// TIA Portal V18 export
// export: Created 2026-06-12T02:00:00Z, ExportSetting WithDefaults, DisplayName Totally Integrated Automation Portal, DisplayVersion V18, DisplayName TIA Portal Openness, DisplayVersion V18
TagTable "AI_B4_Tags"
  AI_B4_Daq_C : Real  (PLC tag AI_B4_Daq_C, HMI_Connection_1, 1 s)   // COUNT 0-100
  AI_B4_TPH_Total : Real  (PLC tag AI_B4_TPH_Total, HMI_Connection_1, 1 s)   // FLOW 100-200 T/h
  AI_B4_KG_CM_Main : Real  (PLC tag AI_B4_KG_CM_Main, HMI_Connection_1, 1 s)   // PRESSURE 7-8 kg/cm2
  AI_B4_DRM_LVL1 : Real  (PLC tag AI_B4_DRM_LVL1, HMI_Connection_1, 1 s)   // LEVEL 30-80 %
  AI_B4_DRM_LVL2 : Real  (PLC tag AI_B4_DRM_LVL2, HMI_Connection_1, 1 s)   // LEVEL 30-80 %
  AI_B4_MW_Output : Real  (PLC tag AI_B4_MW_Output, HMI_Connection_1, 1 s)   // COUNT 0-50 MW
  AI_B4_KG_CM_2 : Real  (PLC tag AI_B4_KG_CM_2, HMI_Connection_1, 1 s)   // PRESSURE 7-8 kg/cm2
  AI_B4_Hc_Value : Real  (PLC tag AI_B4_Hc_Value, HMI_Connection_1, 1 s)   // COUNT 0-100
  AI_B4_Temp_AirHeater_In1 : Real  (PLC tag AI_B4_Temp_AirHeater_In1, HMI_Connection_1, 1 s)   // TEMP 50-80 °C
  AI_B4_Temp_AirHeater_In2 : Real  (PLC tag AI_B4_Temp_AirHeater_In2, HMI_Connection_1, 1 s)   // TEMP 50-80 °C
  AI_B4_Temp_AirHeater_In3 : Real  (PLC tag AI_B4_Temp_AirHeater_In3, HMI_Connection_1, 1 s)   // TEMP 50-80 °C
  AI_B4_Temp_AirHeater_Out1 : Real  (PLC tag AI_B4_Temp_AirHeater_Out1, HMI_Connection_1, 1 s)   // TEMP 50-80 °C
  AI_B4_Temp_AirHeater_Out2 : Real  (PLC tag AI_B4_Temp_AirHeater_Out2, HMI_Connection_1, 1 s)   // TEMP 50-80 °C
  AI_B4_Pres_AH_mmWC_1 : Real  (PLC tag AI_B4_Pres_AH_mmWC_1, HMI_Connection_1, 1 s)   // PRESSURE 7-8 mmWC
  AI_B4_Pres_AH_mmWC_2 : Real  (PLC tag AI_B4_Pres_AH_mmWC_2, HMI_Connection_1, 1 s)   // PRESSURE 7-8 mmWC
  AI_B4_Pres_AH_Pct_1 : Real  (PLC tag AI_B4_Pres_AH_Pct_1, HMI_Connection_1, 1 s)   // PERCENT 20-80 %
  AI_B4_Temp_AH_Out3 : Real  (PLC tag AI_B4_Temp_AH_Out3, HMI_Connection_1, 1 s)   // TEMP 50-80 °C
  AI_B4_Pres_FDH_mmWC : Real  (PLC tag AI_B4_Pres_FDH_mmWC, HMI_Connection_1, 1 s)   // PRESSURE 7-8 mmWC
  AI_B4_RPM_PAF1 : Real  (PLC tag AI_B4_RPM_PAF1, HMI_Connection_1, 1 s)   // RPM 800-1200 RPM
  AI_B4_Pct_RPC308_SP : Real  (PLC tag AI_B4_Pct_RPC308_SP, HMI_Connection_1, 1 s)   // PERCENT 20-80 %
  AI_B4_Pct_RPC308_PV : Real  (PLC tag AI_B4_Pct_RPC308_PV, HMI_Connection_1, 1 s)   // PERCENT 20-80 %
  AI_B4_Pres_PAF1_mmWC : Real  (PLC tag AI_B4_Pres_PAF1_mmWC, HMI_Connection_1, 1 s)   // PRESSURE 7-8 mmWC
  AI_B4_Pct_FDF1_SP : Real  (PLC tag AI_B4_Pct_FDF1_SP, HMI_Connection_1, 1 s)   // PERCENT 20-80 %
  AI_B4_Pct_FDF1_PV : Real  (PLC tag AI_B4_Pct_FDF1_PV, HMI_Connection_1, 1 s)   // PERCENT 20-80 %
  AI_B4_Pct_FDF1_OUT : Real  (PLC tag AI_B4_Pct_FDF1_OUT, HMI_Connection_1, 1 s)   // PERCENT 20-80 %
  AI_B4_RPM_FDF1 : Real  (PLC tag AI_B4_RPM_FDF1, HMI_Connection_1, 1 s)   // RPM 800-1200 RPM
  AI_B4_Pct_RPC301_SP : Real  (PLC tag AI_B4_Pct_RPC301_SP, HMI_Connection_1, 1 s)   // PERCENT 20-80 %
  AI_B4_Pct_RPC301_PV : Real  (PLC tag AI_B4_Pct_RPC301_PV, HMI_Connection_1, 1 s)   // PERCENT 20-80 %
  AI_B4_Pct_RPC301_OUT : Real  (PLC tag AI_B4_Pct_RPC301_OUT, HMI_Connection_1, 1 s)   // PERCENT 20-80 %
  AI_B4_mA_ESP1 : Real  (PLC tag AI_B4_mA_ESP1, HMI_Connection_1, 1 s)   // CURRENT 50-200 mA
  AI_B4_mA_ESP2 : Real  (PLC tag AI_B4_mA_ESP2, HMI_Connection_1, 1 s)   // CURRENT 50-200 mA
  AI_B4_mA_ESP3 : Real  (PLC tag AI_B4_mA_ESP3, HMI_Connection_1, 1 s)   // CURRENT 50-200 mA
  AI_B4_mA_ESP4 : Real  (PLC tag AI_B4_mA_ESP4, HMI_Connection_1, 1 s)   // CURRENT 50-200 mA
  AI_B4_V_ESP1 : Real  (PLC tag AI_B4_V_ESP1, HMI_Connection_1, 1 s)   // COUNT 0-400 V
  AI_B4_V_ESP2 : Real  (PLC tag AI_B4_V_ESP2, HMI_Connection_1, 1 s)   // COUNT 0-400 V
  AI_B4_V_ESP3 : Real  (PLC tag AI_B4_V_ESP3, HMI_Connection_1, 1 s)   // COUNT 0-400 V
  AI_B4_V_ESP4 : Real  (PLC tag AI_B4_V_ESP4, HMI_Connection_1, 1 s)   // COUNT 0-400 V
  AI_B4_Pct_RPC305_SP : Real  (PLC tag AI_B4_Pct_RPC305_SP, HMI_Connection_1, 1 s)   // PERCENT 20-80 %
  AI_B4_Pct_RPC305_PV : Real  (PLC tag AI_B4_Pct_RPC305_PV, HMI_Connection_1, 1 s)   // PERCENT 20-80 %
  AI_B4_RPM_IDF1 : Real  (PLC tag AI_B4_RPM_IDF1, HMI_Connection_1, 1 s)   // RPM 800-1200 RPM
  AI_B4_Pct_RPC305_VFD : Real  (PLC tag AI_B4_Pct_RPC305_VFD, HMI_Connection_1, 1 s)   // PERCENT 20-80 %
  AI_B4_Pct_FDF2_SP : Real  (PLC tag AI_B4_Pct_FDF2_SP, HMI_Connection_1, 1 s)   // PERCENT 20-80 %
  AI_B4_Pct_FDF2_PV : Real  (PLC tag AI_B4_Pct_FDF2_PV, HMI_Connection_1, 1 s)   // PERCENT 20-80 %
  AI_B4_Pct_FDF2_OUT : Real  (PLC tag AI_B4_Pct_FDF2_OUT, HMI_Connection_1, 1 s)   // PERCENT 20-80 %
  AI_B4_RPM_FDF2 : Real  (PLC tag AI_B4_RPM_FDF2, HMI_Connection_1, 1 s)   // RPM 800-1200 RPM
  AI_B4_Pct_RPC306_SP : Real  (PLC tag AI_B4_Pct_RPC306_SP, HMI_Connection_1, 1 s)   // PERCENT 20-80 %
  AI_B4_Pct_RPC306_PV : Real  (PLC tag AI_B4_Pct_RPC306_PV, HMI_Connection_1, 1 s)   // PERCENT 20-80 %
  AI_B4_Pct_RPC306_OUT : Real  (PLC tag AI_B4_Pct_RPC306_OUT, HMI_Connection_1, 1 s)   // PERCENT 20-80 %
  AI_B4_RPM_IDF2 : Real  (PLC tag AI_B4_RPM_IDF2, HMI_Connection_1, 1 s)   // RPM 800-1200 RPM
  AI_B4_Pct_RPC306_VFD : Real  (PLC tag AI_B4_Pct_RPC306_VFD, HMI_Connection_1, 1 s)   // PERCENT 20-80 %
  AI_B4_Pres_FDF_mmWC : Real  (PLC tag AI_B4_Pres_FDF_mmWC, HMI_Connection_1, 1 s)   // PRESSURE 7-8 mmWC
  AI_B4_TEST1_Value : Real  (PLC tag AI_B4_TEST1_Value, HMI_Connection_1, 1 s)   // COUNT 0-100
  AI_B4_Pct_PAF1_SP : Real  (PLC tag AI_B4_Pct_PAF1_SP, HMI_Connection_1, 1 s)   // PERCENT 20-80 %
  AI_B4_Pct_PAF1_PV : Real  (PLC tag AI_B4_Pct_PAF1_PV, HMI_Connection_1, 1 s)   // PERCENT 20-80 %
  AI_B4_Pres_PAF2_mmWC : Real  (PLC tag AI_B4_Pres_PAF2_mmWC, HMI_Connection_1, 1 s)   // PRESSURE 7-8 mmWC
  AI_B4_RPM_PAF2 : Real  (PLC tag AI_B4_RPM_PAF2, HMI_Connection_1, 1 s)   // RPM 800-1200 RPM
  AI_B4_Pct_RPC308b_SP : Real  (PLC tag AI_B4_Pct_RPC308b_SP, HMI_Connection_1, 1 s)   // PERCENT 20-80 %
  AI_B4_Pct_RPC308b_PV : Real  (PLC tag AI_B4_Pct_RPC308b_PV, HMI_Connection_1, 1 s)   // PERCENT 20-80 %
  AI_B4_Pct_DAM303B_SP : Real  (PLC tag AI_B4_Pct_DAM303B_SP, HMI_Connection_1, 1 s)   // PERCENT 20-80 %
  AI_B4_Pct_DAM304B_SP : Real  (PLC tag AI_B4_Pct_DAM304B_SP, HMI_Connection_1, 1 s)   // PERCENT 20-80 %
